(*
  A start position detection function block dummy.
  A dummy implementation to simulate start triggers at desired positions.
  
  NOTE: SubstrateLength can be configured via Job (register I_PrintStatusClien) or directly by property
*)
FUNCTION_BLOCK FB_StartPositionDummy EXTENDS FB_BasePrint IMPLEMENTS I_StartPosDetect, I_PrintStatusClient
VAR_INPUT
  bTrigger                    : BOOL;       // manual trigger
  lPosition                   : DINT;       // current position [SubPx]
  fSpeed                      : LREAL;      // current speed [m/s]
  fResolution                 : LREAL;      // current print resolution [dpi*SubPx]
END_VAR

VAR
  // properties
  _bSim               : BOOL;       // simulatio mode active (PROPERTY)
  _bStartTrig         : BOOL;       // create new CT trigger (PROPERTY)
  _bValid             : BOOL:=TRUE; // (PROPERTY)
  _nStartPosX0        : DINT;       // create position for CT (absolut) [SubPx] (PROPERTY)
  
  // config
  _bAutoTrigger       : BOOL;       // automatic sheet triggers
    
  // local helper
  iJobDefinition      : CalmarCompPrint.I_JobDefinition;
  rfEnable            : RF_TRIG;    // enable edge detection
  rfNewCT             : RF_TRIG;    // start trigger generation
  nSheetLength        : DINT;       // sheet length in [SubPx]
  nSheetGap           : DINT;       // sheet gap in [SubPx]
  nSheetEndPosition   : DINT;       // sheet end position [SubPx]
  nNextSheetPosition  : DINT;       // next trigger location
  fSheetPerHour       : LREAL;      // sheets per hour
  fSheetSpeed         : LREAL;      // [m/min] speed meter per minute
END_VAR

VAR PERSISTENT
  // simulation configuration
  fSheetLength   : LREAL := 0.5;    // [m] sheet length (local or per job given)
  fSheetGap      : LREAL := 0.12;   // [m] gap between two sheets
END_VAR

// checks and fixes
IF iJobDefinition = 0 THEN RETURN; END_IF
IF NOT _bSim THEN RETURN; END_IF
IF fSpeed = 0 THEN RETURN; END_IF
IF fSheetLength = 0 THEN fSheetLength := 1; END_IF
IF fResolution = 0 THEN fResolution := 600*32; END_IF

// calculations
fSheetSpeed := fSpeed * 60;  // [m/s] -> [m/min]
nSheetGap := F_MeterToSubPixel(fPosMeter := fSheetGap, fResoSubPx := fResolution);  // [m] -> [SubPx]
fSheetPerHour := (60*60)/((fSheetLength+fSheetGap)/fSpeed);
nSheetLength := F_MeterToSubPixel(fPosMeter := fSheetLength, fResoSubPx := fResolution);  // [m] -> [SubPx]

rfEnable(CLK:=_bSim);  // initial start at simulation start
IF rfEnable.RT THEN    // start simulation, sample current pos as first X0
  _nStartPosX0 := lPosition;
END_IF

nSheetEndPosition := _nStartPosX0 + nSheetLength;
nNextSheetPosition := nSheetEndPosition + nSheetGap;

// internal trigger creation
IF (lPosition - nNextSheetPosition) > 0 AND _bAutoTrigger THEN
  bTrigger := TRUE;
END_IF

// on trigger
rfNewCT(CLK := bTrigger, RT => _bStartTrig);
IF _bStartTrig THEN
  bTrigger := FALSE;  // reset trigger
  
  _nStartPosX0 := nNextSheetPosition;  // next sheet start position
END_IF

PROPERTY bSimEnable : BOOL
GET
bSimEnable := _bSim;
END_GET
SET
_bSim := bSimEnable;
END_SET
END_PROPERTY

(*
  A new container detected.
  NOTE: a pulse only
*)
PROPERTY bStartTrig : BOOL
GET
bStartTrig := _bStartTrig;
END_GET
END_PROPERTY

(*
  A valid container detected.
*)
PROPERTY bValid : BOOL
GET
bValid := _bValid;
END_GET
END_PROPERTY

PROPERTY fSubstrateLength : LREAL
GET
fSubstrateLength := fSheetLength;
END_GET
SET
fSheetLength := fSubstrateLength;
END_SET
END_PROPERTY

METHOD mJobPause
END_METHOD

METHOD mJobStart
VAR_INPUT
	sJobDef	: CalmarCompPrint.I_JobDefinition;
END_VAR
IF sJobDef = 0 THEN LogError('JobStart: no sJobDef given'); RETURN; END_IF

iJobDefinition := sJobDef;    // current job definition
fSheetLength := iJobDefinition.fSubstrateDepth;
END_METHOD

METHOD mJobStop
VAR_INPUT
	sStatus	: CalmarCompPrint.I_JobStatus;
END_VAR
iJobDefinition := 0;    // delete job definition
END_METHOD

METHOD mProduced
VAR_INPUT
	(* current progress*)
	sProgress	: CalmarCompPrint.I_JobProgress;
END_VAR
; // nothing to do
END_METHOD

(*
  Detected start position X0 (absolute) in [SubPx].
*)
PROPERTY nStartPositionX0 : DINT
GET
nStartPositionX0 := _nStartPosX0;
END_GET
END_PROPERTY

END_FUNCTION_BLOCK

(* stored: Version 1.1.0.1, ProductVersion 3.1.4024.11
   POU FB_StartPositionDummy: Id {6d5938fa-188c-46a3-9614-4d24c87650aa}, SpecialFunc None
   Folder I_PrintStatusClient: Id {1804c86a-7655-4221-b4c5-5f9975e3ba8b}
   Folder I_StartPosDetect: Id {eddb7439-ab58-404f-bfbc-e338b9da7e5a}
   Property bSimEnable: Id {1f412ac1-39c7-4b8e-897a-166f2be0bd7d}
   Get Get: Id {416c9832-37e4-47b9-96b6-19e94cac1c2f}
   Set Set: Id {62a47877-b97c-4288-8caa-d237e4485668}
   Property bStartTrig: Id {ca550c13-f593-4f69-83b3-1db335a17f95}
   Get Get: Id {3d2e4960-ef7b-41e0-ad73-fa3dd64cb60e}
   Property bValid: Id {f9e082ac-9840-4356-b3d4-c6c0e5832b11}
   Get Get: Id {aa86999d-498b-40de-89f4-bdde7f2dd977}
   Property fSubstrateLength: Id {9ca7c39c-2447-4adf-a5db-af2dacbe6d4c}
   Get Get: Id {3ec6aa6f-8875-4f42-b41a-86ee963b8526}
   Set Set: Id {217d62d5-41a6-42e8-a311-44935054e137}
   Method mJobPause: Id {7eb46286-2488-433d-8cdd-400aef51086a}
   Method mJobStart: Id {2e251a78-74c8-4bb3-b07e-90212fae1941}
   Method mJobStop: Id {f5a16969-656a-4350-9777-971b8c8d7ca7}
   Method mProduced: Id {3f03414d-4a1b-4196-a0f6-7c1a726aa09c}
   Property nStartPositionX0: Id {e2effe83-ef6c-4a3b-86b8-29a14d846434}
   Get Get: Id {5e8f9341-de59-4c4a-8866-59b0baf4f592} *)
